// Mitsubishi GX Works2 project: 연속동작   PLC: Q02/Q02H

PROGRAM MAIN
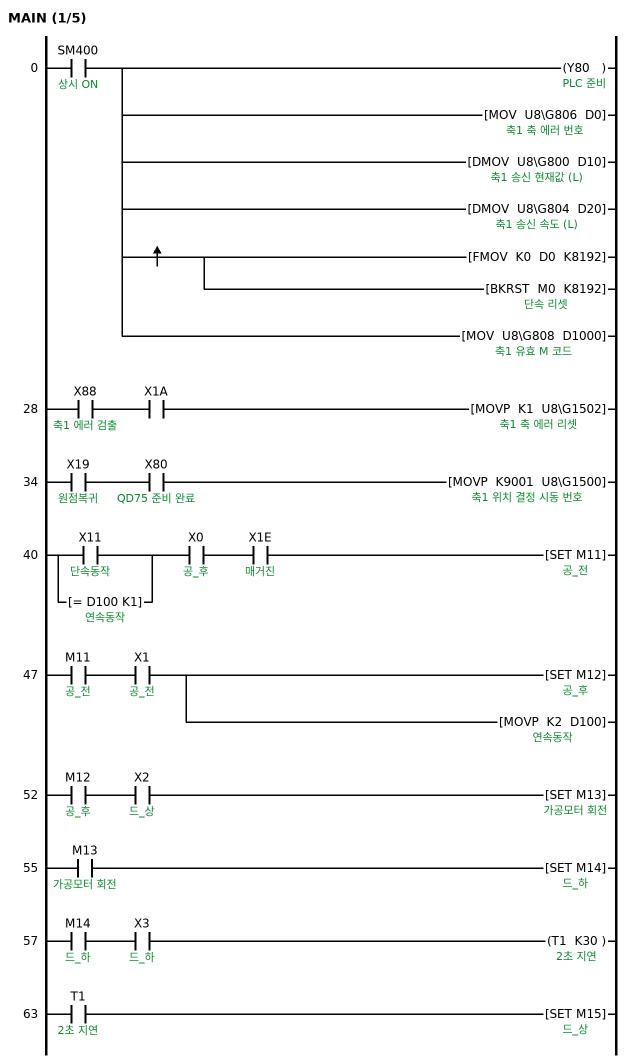
0     LD      SM400  ; 상시 ON
      OUT     Y80  ; PLC 준비
      MOV     U8\G806 D0  ; 축1 축 에러 번호
      DMOV    U8\G800 D10  ; 축1 송신 현재값 (L)
      DMOV    U8\G804 D20  ; 축1 송신 속도 (L)
      MPS
      MEP
      FMOV    K0 D0 K8192
      BKRST   M0 K8192  ; 단속 리셋
      MPP
      MOV     U8\G808 D1000  ; 축1 유효 M 코드
28    LD      X88  ; 축1 에러 검출
      AND     X1A
      MOVP    K1 U8\G1502  ; 축1 축 에러 리셋
34    LD      X19  ; 원점복귀
      AND     X80  ; QD75 준비 완료
      MOVP    K9001 U8\G1500  ; 축1 위치 결정 시동 번호
40    LD      X11  ; 단속동작
      OR=     D100 K1  ; 연속동작
      AND     X0  ; 공_후
      AND     X1E  ; 매거진
      SET     M11  ; 공_전
47    LD      M11  ; 공_전
      AND     X1  ; 공_전
      SET     M12  ; 공_후
      MOVP    K2 D100
52    LD      M12  ; 공_후
      AND     X2  ; 드_상
      SET     M13  ; 가공모터 회전
55    LD      M13  ; 가공모터 회전
      SET     M14  ; 드_하
57    LD      M14  ; 드_하
      AND     X3  ; 드_하
      OUT     T1 K30  ; 2초 지연
63    LD      T1  ; 2초 지연
      SET     M15  ; 드_상
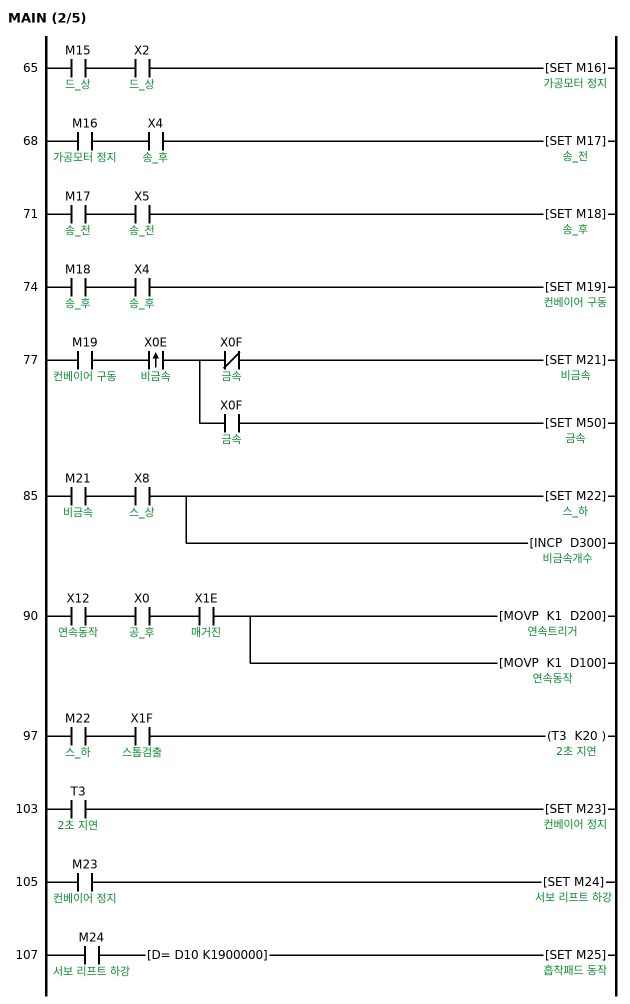
65    LD      M15  ; 드_상
      AND     X2  ; 드_상
      SET     M16  ; 가공모터 정지
68    LD      M16  ; 가공모터 정지
      AND     X4  ; 송_후
      SET     M17  ; 송_전
71    LD      M17  ; 송_전
      AND     X5  ; 송_전
      SET     M18  ; 송_후
74    LD      M18  ; 송_후
      AND     X4  ; 송_후
      SET     M19  ; 컨베이어 구동
77    LD      M19  ; 컨베이어 구동
      ANDP    X0E  ; 비금속
      MPS
      ANI     X0F  ; 금속
      SET     M21  ; 비금속
      MPP
      AND     X0F  ; 금속
      SET     M50  ; 금속
85    LD      M21  ; 비금속
      AND     X8  ; 스_상
      SET     M22  ; 스_하
      INCP    D300  ; 비금속개수
90    LD      X12  ; 연속동작
      AND     X0  ; 공_후
      AND     X1E  ; 매거진
      MOVP    K1 D200  ; 연속트리거
      MOVP    K1 D100
97    LD      M22  ; 스_하
      AND     X1F  ; 스톱검출
      OUT     T3 K20  ; 2초 지연
103   LD      T3  ; 2초 지연
      SET     M23  ; 컨베이어 정지
105   LD      M23  ; 컨베이어 정지
      SET     M24  ; 서보 리프트 하강
107   LD      M24  ; 서보 리프트 하강
      ANDD=   D10 K1900000
      SET     M25  ; 흡착패드 동작
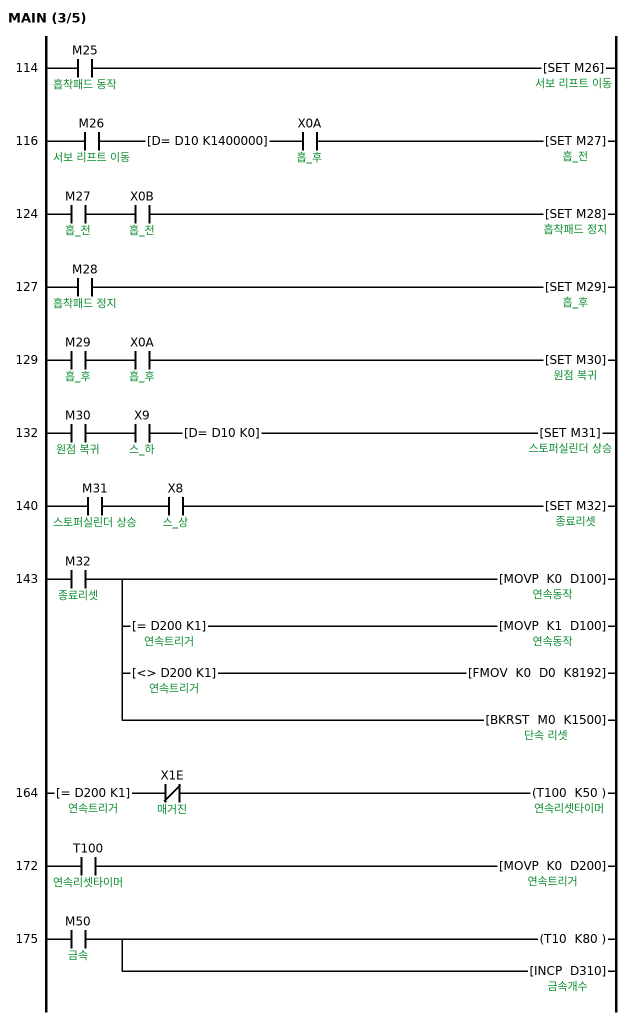
114   LD      M25  ; 흡착패드 동작
      SET     M26  ; 서보 리프트 이동
116   LD      M26  ; 서보 리프트 이동
      ANDD=   D10 K1400000
      AND     X0A  ; 흡_후
      SET     M27  ; 흡_전
124   LD      M27  ; 흡_전
      AND     X0B  ; 흡_전
      SET     M28  ; 흡착패드 정지
127   LD      M28  ; 흡착패드 정지
      SET     M29  ; 흡_후
129   LD      M29  ; 흡_후
      AND     X0A  ; 흡_후
      SET     M30  ; 원점 복귀
132   LD      M30  ; 원점 복귀
      AND     X9  ; 스_하
      ANDD=   D10 K0
      SET     M31  ; 스토퍼실린더 상승
140   LD      M31  ; 스토퍼실린더 상승
      AND     X8  ; 스_상
      SET     M32  ; 종료리셋
143   LD      M32  ; 종료리셋
      MOVP    K0 D100
      MPS
      AND=    D200 K1  ; 연속트리거
      MOVP    K1 D100
      MRD
      AND<>   D200 K1  ; 연속트리거
      FMOV    K0 D0 K8192
      MPP
      BKRST   M0 K1500
164   LD=     D200 K1  ; 연속트리거
      ANI     X1E  ; 매거진
      OUT     T100 K50  ; 연속리셋타이머
172   LD      T100  ; 연속리셋타이머
      MOVP    K0 D200
175   LD      M50  ; 금속
      OUT     T10 K80
      INCP    D310  ; 금속개수
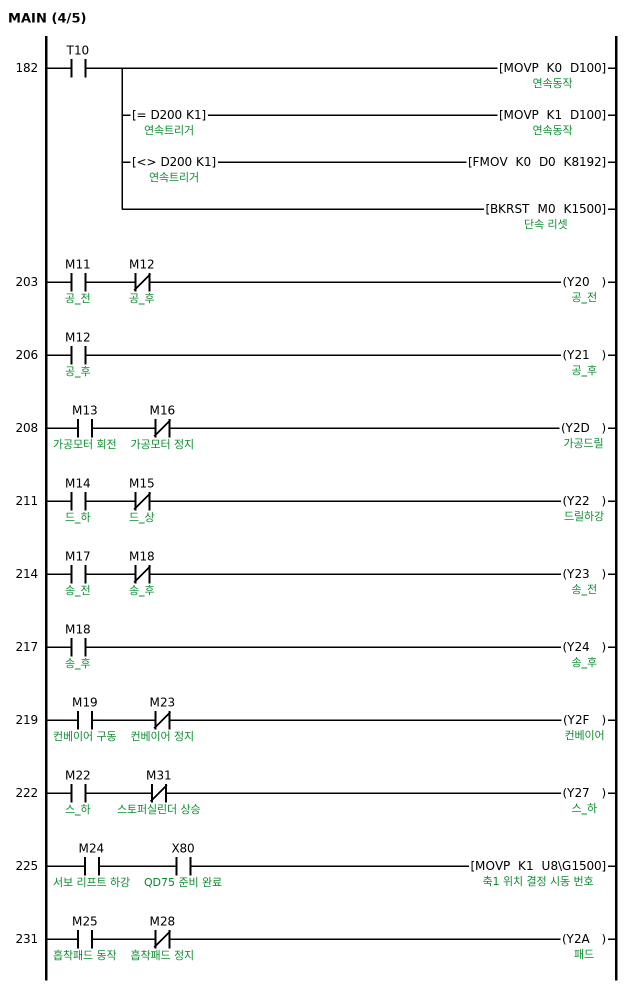
182   LD      T10
      MOVP    K0 D100
      MPS
      AND=    D200 K1  ; 연속트리거
      MOVP    K1 D100
      MRD
      AND<>   D200 K1  ; 연속트리거
      FMOV    K0 D0 K8192
      MPP
      BKRST   M0 K1500
203   LD      M11  ; 공_전
      ANI     M12  ; 공_후
      OUT     Y20  ; 공_전
206   LD      M12  ; 공_후
      OUT     Y21  ; 공_후
208   LD      M13  ; 가공모터 회전
      ANI     M16  ; 가공모터 정지
      OUT     Y2D  ; 가공드릴
211   LD      M14  ; 드_하
      ANI     M15  ; 드_상
      OUT     Y22  ; 드릴하강
214   LD      M17  ; 송_전
      ANI     M18  ; 송_후
      OUT     Y23  ; 송_전
217   LD      M18  ; 송_후
      OUT     Y24  ; 송_후
219   LD      M19  ; 컨베이어 구동
      ANI     M23  ; 컨베이어 정지
      OUT     Y2F  ; 컨베이어
222   LD      M22  ; 스_하
      ANI     M31  ; 스토퍼실린더 상승
      OUT     Y27  ; 스_하
225   LD      M24  ; 서보 리프트 하강
      AND     X80  ; QD75 준비 완료
      MOVP    K1 U8\G1500
231   LD      M25  ; 흡착패드 동작
      ANI     M28  ; 흡착패드 정지
      OUT     Y2A  ; 패드
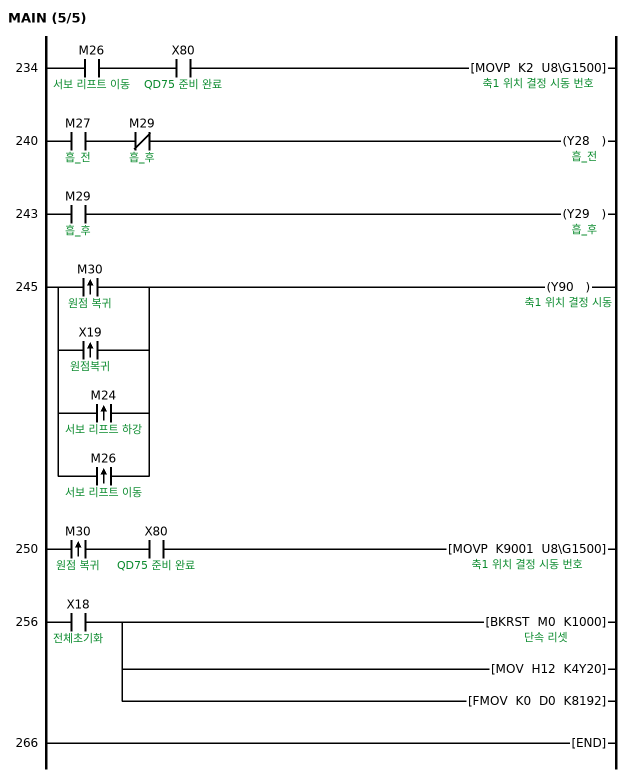
234   LD      M26  ; 서보 리프트 이동
      AND     X80  ; QD75 준비 완료
      MOVP    K2 U8\G1500
240   LD      M27  ; 흡_전
      ANI     M29  ; 흡_후
      OUT     Y28  ; 흡_전
243   LD      M29  ; 흡_후
      OUT     Y29  ; 흡_후
245   LDP     M30  ; 원점 복귀
      ORP     X19  ; 원점복귀
      ORP     M24  ; 서보 리프트 하강
      ORP     M26  ; 서보 리프트 이동
      OUT     Y90  ; 축1 위치 결정 시동
250   LDP     M30  ; 원점 복귀
      AND     X80  ; QD75 준비 완료
      MOVP    K9001 U8\G1500
256   LD      X18  ; 전체초기화
      BKRST   M0 K1000
      MOV     H12 K4Y20
      FMOV    K0 D0 K8192
266   END
END_PROGRAM

// device comments not shown above
X6  ; 배_후
X7  ; 배_전
X0C  ; 창_후
X0D  ; 창_전
X10  ; 매거진
X13  ; 종료
X81  ; 동기용 플래그
X84  ; 축1 M 코드 ON
X85  ; 축2 M 코드 ON
X89  ; 축2 에러 검출
X8C  ; 축1 BUSY
X8D  ; 축2 BUSY
X90  ; 축1 시동 완료
X91  ; 축2 시동 완료
X94  ; 축1 위치 결정 완료
X95  ; 축2 위치 결정 완료
Y25  ; 배_전
Y26  ; 배_후
Y2B  ; 창_전
Y2C  ; 창_후
Y84  ; 축1 축 정지
Y85  ; 축2 축 정지
Y88  ; 축1 정운전 JOG 시동
Y89  ; 축1 역운전 JOG 시동
Y8A  ; 축2 정운전 JOG 시동
Y8B  ; 축2 역운전 JOG 시동
Y91  ; 축2 위치 결정 시동
Y94  ; 축1 실행 금지 플래그
Y95  ; 축2 실행 금지 플래그
M20  ; 동작끝
M100  ; 연속동작
M101  ; 연속동작 종료
M200  ; 연속동작 금속
M300  ; 연속동작 비금속
M800  ; 연속리셋
M1000  ; 연속시작
M1500  ; 연속시작
M1900  ; 연속리셋
T2  ; 8초 동작
